// Interface for digital IO
INTERFACE I_DIO

// Run this method every cycle
METHOD ABSTRACT Execute
END_METHOD

// Get the name of the IO
PROPERTY Name : STRING
GET
END_GET
END_PROPERTY

END_INTERFACE

(* stored: Version 1.1.0.1, ProductVersion 3.1.4024.11
   Itf I_DIO: Id {f1581428-788b-4a2e-a426-fff7782cd4db}
   Folder Methods: Id {9cc62082-6678-4dc2-8906-2fc64b040f55}
   Folder Properties: Id {2285bdb0-d2fe-445c-88c0-8c1800a2bf09}
   Method Execute: Id {19c37d63-a0b5-41d5-9859-121985fbaeb0}
   Property Name: Id {3753ce80-58b9-481d-bd97-aa8e15fad4a9}
   Get Get: Id {d3a00ebc-7e08-44c2-a232-f3d21957063e} *)
